ABB RobotStudio station: Estacio120_ROBOTARI_G9.rspag

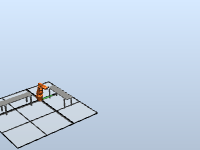
--- station ---
Station Estacio120_ROBOTARI_1415 (saved by RobotStudio format 3)
Controller Sistema120_LEGO_CLOT
  mechanical unit ROB_1: IRB120_3_58__01, 6 joints, base frame (0, 0, 0) mm
Layout (positions relative to the parent item):
  - IRB120_3_58__01 [mechanism, from Robots\IRB120_3_58__01.rslib] at (0, 0, 0) mm; joint values [0.119, 0.2462, -0.2116, 0.435, 0.1998, -0.6575] (rad or m)
  - VENTOSA [mechanism] at (436.31, 58.24, 595.96) mm, rotated rx -12.13 ry 12.35 rz 11.73 deg
      TCP VENTOSA at (0, 0, 0) mm
      links: Conjunto ventosa-muñon
  - Cinta_1 [part] at (0, -1110, 367) mm, rotated rx 0 ry 0 rz 90 deg
  - CINTA2 [part] at (575, 475, 400) mm
Attachment: VENTOSA is attached to IRB120_3_58__01 / Link6
Collision set Conjunto de colisión_1: IRB120_3_58__01, VENTOSA against CINTA2, Cinta_1, near miss 0 m

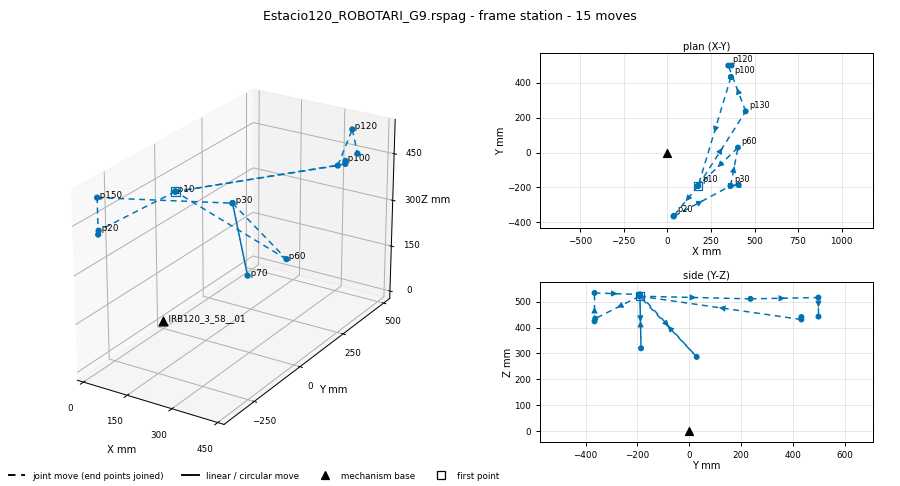
[picture p0: tool path of Estacio120_ROBOTARI_G9.rspag in frame station, 15 of 19 moves have a stored position in this frame; points joined in program order, loops and branches not executed]
--- Backups/Sistema120_LEGO_CLOT/RAPID/TASK1/PROGMOD/CalibData.mod ---
MODULE CalibData
	PERS tooldata VENTOSA:=[TRUE,[[0,0,0],[0.707106781,0,-0.707106781,0]],[0.2,[-60,47,25],[1,0,0,0],0,0,0]];
	TASK PERS tooldata Toolventosa_1:=[TRUE,[[70,0,40],[0.707106781,0,-0.707106781,0]],[0.2,[10,20,10],[1,0,0,0],0,0,0]];
ENDMODULE

--- Backups/Sistema120_LEGO_CLOT/RAPID/TASK1/PROGMOD/MainModule.mod ---
MODULE MainModule

    CONST jointtarget jpos10:=[[6.81954,14.1088,-12.1243,24.9211,11.4493,-37.6717],[9E+09,9E+09,9E+09,9E+09,9E+09,9E+09]];
	CONST robtarget p10:=[[176.81,-191.57,521.21],[0.278921,-0.372832,-0.862871,-0.196606],[-1,0,-1,0],[9E+09,9E+09,9E+09,9E+09,9E+09,9E+09]];
	CONST robtarget p20:=[[36.45,-363.29,434.61],[0.151188,-0.68875,-0.66446,-0.247506],[-1,0,-1,1],[9E+09,9E+09,9E+09,9E+09,9E+09,9E+09]];
	CONST robtarget p30:=[[362.93,-190.78,527.78],[0.208623,-0.296741,-0.924245,-0.119128],[-1,0,-1,1],[9E+09,9E+09,9E+09,9E+09,9E+09,9E+09]];
	CONST robtarget p40:=[[403.50,-186.18,39.16],[0.220229,-0.193089,-0.950068,-0.107642],[-1,-1,0,1],[9E+09,9E+09,9E+09,9E+09,9E+09,9E+09]];
	CONST robtarget p50:=[[405.19,32.89,41.83],[0.208965,-0.192578,-0.952954,-0.105477],[0,0,0,1],[9E+09,9E+09,9E+09,9E+09,9E+09,9E+09]];
	CONST robtarget p60:=[[405.02,28.65,286.65],[0.210569,-0.192705,-0.952533,-0.105863],[0,0,-1,1],[9E+09,9E+09,9E+09,9E+09,9E+09,9E+09]];
	CONST robtarget p70:=[[408.73,-186.25,320.05],[0.21057,-0.192707,-0.952533,-0.105858],[-1,-1,0,1],[9E+09,9E+09,9E+09,9E+09,9E+09,9E+09]];
	CONST robtarget p80:=[[182.80,243.44,681.59],[0.239987,0.420452,-0.872058,0.0716986],[0,0,-1,0],[9E+09,9E+09,9E+09,9E+09,9E+09,9E+09]];
	CONST robtarget p90:=[[364.78,432.80,431.28],[0.29221,0.277543,-0.915161,-0.00793556],[0,-2,1,0],[9E+09,9E+09,9E+09,9E+09,9E+09,9E+09]];
	CONST robtarget p100:=[[364.79,432.79,440.77],[0.292242,0.277494,-0.915166,-0.00792924],[0,-2,1,0],[9E+09,9E+09,9E+09,9E+09,9E+09,9E+09]];
	CONST robtarget p110:=[[368.76,498.78,442.48],[0.292218,0.277507,-0.91517,-0.00789908],[0,-2,1,0],[9E+09,9E+09,9E+09,9E+09,9E+09,9E+09]];
	CONST robtarget p120:=[[349.63,498.54,515.95],[0.262768,0.480674,-0.835673,0.0394526],[0,0,-1,0],[9E+09,9E+09,9E+09,9E+09,9E+09,9E+09]];
	CONST robtarget p130:=[[449.31,236.18,510.99],[0.369937,0.152754,-0.914397,0.0607572],[0,-1,0,0],[9E+09,9E+09,9E+09,9E+09,9E+09,9E+09]];
    CONST robtarget p140:=[[36.47,-365.92,423.85],[0.138204,-0.694353,-0.66549,-0.236425],[-1,0,-1,1],[9E+09,9E+09,9E+09,9E+09,9E+09,9E+09]];
   	CONST robtarget p150:=[[36.44,-365.93,533.78],[0.138198,-0.694384,-0.665464,-0.236409],[-1,0,-1,1],[9E+09,9E+09,9E+09,9E+09,9E+09,9E+09]];
   	LOCAL VAR num Fila_COM1:=0;
   	LOCAL VAR num Columna_COM1:=0;
   	LOCAL VAR num Fila_COM2:=0;
    LOCAL VAR num Columna_COM2:=0;
   	LOCAL VAR bool COM:=False;
    LOCAL VAR bool Peça:=False;
    LOCAL VAR bool Primera_peça:=False;



 PROC  COMANDA(num Columna,num Fila,bool COM)

     FOR Files FROM 0 TO Fila DO

         FOR Columnes FROM 0 TO Columna DO

             IF COM=TRUE THEN

                    MoveJ Offs (p50,(Fila*37.5),(Columna*37.5),0), v1000, fine, tool_ventosa;

             ELSEIF  COM=FALSE THEN

                    MoveJ Offs (p40,(Fila*37.5),(Columna*37.5),0), v1000, fine, tool_ventosa;
             ENDIF
     ENDFOR
        ENDFOR
 ENDPROC



	PROC main()

   !Reset DO10_3;
   SetDO DO10_1,1;  !Activar el compressor
   !POSICIO DE INICI
     MoveAbsJ jpos10\NoEOffs, v1000, z50, tool_ventosa;



 !Espera ordre de final de cicle------------------------------------------------------------------------------------
    IF DI10_4=1 OR Primera_peça=False THEN

     WaitDI DI10_1,1;
     !POSICIO DE LA CINTA 1 ON ESTA LA PEÇA
     MoveJ p10, v1000, z0, tool_ventosa;
     MoveJ p20, v1000, z0, tool_ventosa;
     SetDO DO10_2,1;
     Reset DO10_3;
     MoveJ p140, v1000, z0, tool_ventosa;
     MoveJ p150, v1000, fine, tool_ventosa;
     Peça:=True;
     Primera_peça:=FALSE;

    ENDIF
!Ordre al robot enviar peça a la Comanda 1------------------------------------------------------------------------------------

   IF DI10_2=0 AND  DI10_3=0 AND Peça  THEN      !00

    COM:=False;

   IF Columna_COM1>4 THEN
    Add Fila_COM1,1;
    Columna_COM1:=0;
    ENDIF

    IF Fila_COM1>4 THEN
       Fila_COM1:=0;
    ENDIF

   MoveJ p30, v1000, z0, tool_ventosa;
   MoveJ p70, v1000, z0, tool_ventosa;
   !POSICIO DE LA COMANDA 1
   COMANDA Columna_COM1,Fila_COM1,COM;
   Add Columna_COM1,1;
   Reset DO10_2;
   SetDO DO10_3,1;
   Peça:=False;

   ENDIF

!Ordre al robot enviar peça a la Comanda 2------------------------------------------------------------------------------------

    IF  DI10_2=0 AND  DI10_3=1 AND Peça THEN         !01

    COM:=True;
    IF Columna_COM2>4 THEN
       Add Fila_COM2,1;
       Columna_COM2:=0;
    ENDIF

     IF Fila_COM2>4 THEN
       Fila_COM2:=0;
    ENDIF

    MoveJ p30, v1000, z0, tool_ventosa;
    MoveJ p60, v1000, z0, tool_ventosa;
    !POSICIO DE LA COMANDA 2
    COMANDA Columna_COM2,Fila_COM2,COM;
    Add Columna_COM2,1;
    Reset DO10_2;
    SetDO DO10_3,1;
    Peça:=False;

    ENDIF

!Ordre al robot enviar peça a la cinta 2 a la primera posició------------------------------------------------------------------------------------

    IF  DI10_2=1 AND DI10_3=0 AND Peça THEN        !10
        !POSICIO DEL MAGATZEM 1-2
        MoveJ p10, v1000, z0, tool_ventosa;
        MoveAbsJ jpos10\NoEOffs, v1000, z50, tool_ventosa;
        MoveJ p100, v1000, z0, tool_ventosa;
        MoveL p90, v1000, z0, tool_ventosa;
        Reset DO10_2;
        SetDO DO10_3,1;
        Peça:=False;
        Primera_peça:=True;

    ENDIF

!Ordre al robot enviar peça a la cinta 2 a la segona posició------------------------------------------------------------------------------------

    IF  DI10_2=1 AND  DI10_3=1 AND Peça THEN            !11
        !POSICIO DEL MAGATZEM 3-4
         MoveJ p10, v1000, z0, tool_ventosa;
         MoveJ p130, v1000, z0, tool_ventosa;
         MoveJ p120, v1000, z0, tool_ventosa;
         MoveJ p110, v1000, z0, tool_ventosa;
        Reset DO10_2;
        SetDO DO10_3,1;
        Peça:=False;
        Primera_peça:=True;

    ENDIF



	ENDPROC
ENDMODULE

--- Backups/Sistema120_LEGO_CLOT/HOME/NewProgramName/MainModule.mod ---
MODULE MainModule
	PROC main()

	ENDPROC
ENDMODULE

--- Backups/Sistema120_LEGO_CLOT/SYSPAR/EIO.cfg ---
EIO:CFG_1.0:5:0::
#
EIO_BUS:

      -Name "Virtual1" -ConnectorID "SIM1"

      -Name "DeviceNet1" -BusType "DNET" -ConnectorID "PCI1"\
      -ConnectorLabel "First DeviceNet"

      -Name "DeviceNet_Lean" -BusType "DNLE" -ConnectorID "PCI1"\
      -ConnectorLabel "DeviceNet Lean"

      -Name "Profinet1" -BusType "PNET" -ConnectorID "PCI1"
#
EIO_UNIT_TYPE:

      -Name "Virtual" -VendorName "ABB" -ProductName "Virtual unit"

      -Name "DN_GENERIC" -BusType "DNET" -DN_ExplicitMsgEnabled \
      -DN_C1OutputSize -1 -DN_C1InputSize -1

      -Name "d320" -BusType "DNET" -VendorName "ABB Robotics"\
      -ProductName "120 Vac Unit" -DN_VendorId 75 -DN_ProductCode 1\
      -DN_DeviceType 7 -DN_MajorRev 1 -DN_ExplicitMsgEnabled  -DN_C1Interval 50\
      -DN_C1OutputSize 2 -DN_C1InputSize 2

      -Name "d327A" -BusType "DNET" -VendorName "ABB Robotics"\
      -ProductName "Combi Unit" -DN_VendorId 75 -DN_ProductCode 2\
      -DN_DeviceType 100 -DN_MajorRev 5 -DN_ExplicitMsgEnabled  -DN_C1Type "COS"\
      -DN_C1OutputSize 6 -DN_C1InputSize 2

      -Name "d328A" -BusType "DNET" -VendorName "ABB Robotics"\
      -ProductName "24 VDC Unit" -DN_VendorId 75 -DN_ProductCode 3\
      -DN_DeviceType 7 -DN_ExplicitMsgEnabled  -DN_C1Type "COS"\
      -DN_C1OutputSize 2 -DN_C1InputSize 2

      -Name "d332A" -BusType "DNET" -VendorName "ABB Robotics"\
      -ProductName "Relay Unit" -DN_VendorId 75 -DN_ProductCode 5\
      -DN_DeviceType 7 -DN_MajorRev 2 -DN_ExplicitMsgEnabled  -DN_C1Type "COS"\
      -DN_C1OutputSize 2 -DN_C1InputSize 2

      -Name "d355A" -BusType "DNET" -VendorName "ABB Robotics"\
      -ProductName "Analog Unit" -DN_VendorId 75 -DN_ProductCode 10\
      -DN_DeviceType 100 -DN_MajorRev 1 -DN_ExplicitMsgEnabled \
      -DN_C1Interval 50 -DN_C1OutputSize 8 -DN_C1InputSize 8

      -Name "d651" -BusType "DNET" -VendorName "ABB Robotics"\
      -ProductName "Combi Unit" -DN_VendorId 75 -DN_ProductCode 25\
      -DN_DeviceType 100 -DN_ExplicitMsgEnabled  -DN_C1Type "COS"\
      -DN_C1OutputSize 5 -DN_C1InputSize 1

      -Name "d652" -BusType "DNET" -VendorName "ABB Robotics"\
      -ProductName "24 VDC Unit" -DN_VendorId 75 -DN_ProductCode 26\
      -DN_DeviceType 7 -DN_ExplicitMsgEnabled  -DN_C1Type "COS"\
      -DN_C1OutputSize 2 -DN_C1InputSize 2

      -Name "d653" -BusType "DNET" -VendorName "ABB Robotics"\
      -ProductName "Relay Unit" -DN_VendorId 75 -DN_ProductCode 27\
      -DN_DeviceType 7 -DN_ExplicitMsgEnabled  -DN_C1Type "COS"\
      -DN_C1OutputSize 1 -DN_C1InputSize 1

      -Name "DN_SLAVE" -BusType "DNET" -VendorName "ABB Robotics" -DN_VendorId 8\
      -DN_ProductCode 12 -DN_DeviceType 12 -DN_ExplicitMsgEnabled \
      -DN_C1Interval 50 -DN_C1OutputSize 8 -DN_C1InputSize 8

      -Name "DN_INTERNAL_SLAVE" -BusType "DNET" -VendorName "ABB Robotics"\
      -ProductName "Internal DeviceNet Slave" -InternalSlave  -DN_C1OutputSize 8\
      -DN_C1InputSize 8

      -Name "d350B" -BusType "DNET" -VendorName "ABB Robotics"\
      -ProductName "RIO Adapter" -DN_VendorId 75 -DN_ProductCode 6\
      -DN_DeviceType 7 -DN_MajorRev 2 -DN_ExplicitMsgEnabled  -DN_C1Type "COS"\
      -DN_C1OutputSize -1 -DN_C1InputSize -1

      -Name "d351A" -BusType "DNET" -VendorName "ABB Robotics"\
      -ProductName "IBS Adapter" -DN_VendorId 75 -DN_ProductCode 7\
      -DN_DeviceType 7 -DN_MajorRev 1 -DN_ExplicitMsgEnabled  -DN_C1Type "COS"\
      -DN_C1OutputSize -1 -DN_C1InputSize -1

      -Name "d352A" -BusType "DNET" -VendorName "ABB Robotics"\
      -ProductName "PBUS Adapter" -DN_VendorId 75 -DN_ProductCode 8\
      -DN_DeviceType 7 -DN_MajorRev 1 -DN_ExplicitMsgEnabled  -DN_C1Type "COS"\
      -DN_C1OutputSize -1 -DN_C1InputSize -1

      -Name "d352B" -BusType "DNET" -VendorName "ABB Robotics"\
      -ProductName "PBUS Adapter" -DN_VendorId 75 -DN_ProductCode 8\
      -DN_DeviceType 7 -DN_MajorRev 1 -DN_ExplicitMsgEnabled  -DN_C1Type "COS"\
      -DN_C1OutputSize -1 -DN_C1InputSize -1

      -Name "d378A" -BusType "DNET" -VendorName "ABB Robotics"\
      -ProductName "CCLink Adapter" -DN_VendorId 75 -DN_ProductCode 17\
      -DN_DeviceType 7 -DN_MajorRev 1 -DN_ExplicitMsgEnabled  -DN_C1Interval 50\
      -DN_C1OutputSize -1 -DN_C1InputSize -1

      -Name "d651_Lean" -BusType "DNLE" -VendorName "ABB Robotics"\
      -ProductName "Combi Unit" -DL_ProductCode 25

      -Name "d652_Lean" -BusType "DNLE" -VendorName "ABB Robotics"\
      -ProductName "24 VDC Unit" -DL_ProductCode 26

      -Name "d653_Lean" -BusType "DNLE" -VendorName "ABB Robotics"\
      -ProductName "Relay Unit" -DL_ProductCode 27

      -Name "AC500_PLC_Lean" -BusType "DNLE" -VendorName "ABB Stotz"\
      -ProductName "AC500 PLC - FPB" -DL_ProductCode 1 -DL_VendorID 760

      -Name "DL_GENERIC" -BusType "DNLE" -DL_ProductCode 3535

      -Name "DL_GENERIC_POLL" -BusType "DNLE" -DL_ProductCode 3535\
      -DL_Pollrate 30

      -Name "d351_Lean" -BusType "DNLE" -VendorName "ABB Robotics"\
      -ProductName "IBS Adapter" -DL_ProductCode 7

      -Name "d352_Lean" -BusType "DNLE" -VendorName "ABB Robotics"\
      -ProductName "PBUS Adapter" -DL_ProductCode 8

      -Name "d378_Lean" -BusType "DNLE" -VendorName "ABB Robotics"\
      -ProductName "CCLink Adapter" -DL_ProductCode 17

      -Name "PN_GENERIC" -BusType "PNET" -ProductName "Profinet Device"

      -Name "PN_INTERNAL_SLAVE" -BusType "PNET" -VendorName "ABB Robotics"\
      -ProductName "Internal Profinet Slave" -InternalSlave
#
EIO_UNIT:

      -Name "D652_10" -UnitType "d652" -Bus "DeviceNet1" -DN_Address 10
#
EIO_SIGNAL:

      -Name "DI10_1" -SignalType "DI" -Unit "D652_10" -UnitMap "0"

      -Name "DI10_2" -SignalType "DI" -Unit "D652_10" -UnitMap "1"

      -Name "DI10_3" -SignalType "DI" -Unit "D652_10" -UnitMap "2"

      -Name "DI10_4" -SignalType "DI" -Unit "D652_10" -UnitMap "3"

      -Name "DI10_5" -SignalType "DI" -Unit "D652_10" -UnitMap "4"

      -Name "DI10_6" -SignalType "DI" -Unit "D652_10" -UnitMap "5"

      -Name "DI10_7" -SignalType "DI" -Unit "D652_10" -UnitMap "6"

      -Name "DI10_8" -SignalType "DI" -Unit "D652_10" -UnitMap "7"

      -Name "DI10_9" -SignalType "DI" -Unit "D652_10" -UnitMap "8"

      -Name "DI10_10" -SignalType "DI" -Unit "D652_10" -UnitMap "9"

      -Name "DI10_11" -SignalType "DI" -Unit "D652_10" -UnitMap "10"

      -Name "DI10_12" -SignalType "DI" -Unit "D652_10" -UnitMap "11"

      -Name "DI10_13" -SignalType "DI" -Unit "D652_10" -UnitMap "12"

      -Name "DI10_14" -SignalType "DI" -Unit "D652_10" -UnitMap "13"

      -Name "DI10_15" -SignalType "DI" -Unit "D652_10" -UnitMap "14"

      -Name "DI10_16" -SignalType "DI" -Unit "D652_10" -UnitMap "15"

      -Name "DO10_1" -SignalType "DO" -Unit "D652_10" -UnitMap "0"

      -Name "DO10_2" -SignalType "DO" -Unit "D652_10" -UnitMap "1"

      -Name "DO10_3" -SignalType "DO" -Unit "D652_10" -UnitMap "2"

      -Name "DO10_4" -SignalType "DO" -Unit "D652_10" -UnitMap "3"

      -Name "DO10_5" -SignalType "DO" -Unit "D652_10" -UnitMap "4"

      -Name "DO10_6" -SignalType "DO" -Unit "D652_10" -UnitMap "5"

      -Name "DO10_7" -SignalType "DO" -Unit "D652_10" -UnitMap "6"

      -Name "DO10_8" -SignalType "DO" -Unit "D652_10" -UnitMap "7"

      -Name "DO10_9" -SignalType "DO" -Unit "D652_10" -UnitMap "8"

      -Name "DO10_10" -SignalType "DO" -Unit "D652_10" -UnitMap "9"

      -Name "DO10_11" -SignalType "DO" -Unit "D652_10" -UnitMap "10"

      -Name "DO10_12" -SignalType "DO" -Unit "D652_10" -UnitMap "11"

      -Name "DO10_13" -SignalType "DO" -Unit "D652_10" -UnitMap "12"

      -Name "DO10_14" -SignalType "DO" -Unit "D652_10" -UnitMap "13"

      -Name "DO10_15" -SignalType "DO" -Unit "D652_10" -UnitMap "14"

      -Name "DO10_16" -SignalType "DO" -Unit "D652_10" -UnitMap "15"
#
EIO_COMMAND_TYPE:

      -Name "LinkAddr" -UnitType "d350B" -DefValue "1" -OrderNr 1\
      -DN_Path "6,20 64 24 01 30 01,C6,1" -DN_Service 16

      -Name "DataRate" -UnitType "d350B" -DefValue "0" -OrderNr 2\
      -DN_Path "6,20 64 24 01 30 02,C6,1" -DN_Service 16

      -Name "StartQ" -UnitType "d350B" -DefValue "0" -OrderNr 3\
      -DN_Path "6,20 64 24 01 30 03,C6,1" -DN_Service 16

      -Name "RackSize" -UnitType "d350B" -DefValue "0" -OrderNr 4\
      -DN_Path "6,20 64 24 01 30 04,C6,1" -DN_Service 16

      -Name "LastRack" -UnitType "d350B" -DefValue "0" -OrderNr 5\
      -DN_Path "6,20 64 24 01 30 05,C1,1" -DN_Service 16

      -Name "D350Breset" -UnitType "d350B" -DefValue "0" -OrderNr 6\
      -DN_Path "4,20 01 24 01,C1,1" -DN_Service 5

      -Name "DataWidth" -UnitType "d351A" -DefValue "3" -OrderNr 1\
      -DN_Path "6,20 65 24 01 30 01,C6,1" -DN_Service 16

      -Name "D351Areset" -UnitType "d351A" -DefValue "0" -OrderNr 2\
      -DN_Path "4,20 01 24 01,C1,1" -DN_Service 5

      -Name "MasterInputSize" -UnitType "d352A" -DefValue "1" -OrderNr 1\
      -DN_Path "6,20 67 24 01 30 02,C6,1" -DN_Service 16

      -Name "MasterOutputSize" -UnitType "d352A" -DefValue "1" -OrderNr 2\
      -DN_Path "6,20 67 24 01 30 03,C6,1" -DN_Service 16

      -Name "StationAddress" -UnitType "d352A" -DefValue "126" -OrderNr 3\
      -DN_Path "6,20 67 24 01 30 04,C6,1" -DN_Service 16

      -Name "D352Areset" -UnitType "d352A" -DefValue "0" -OrderNr 4\
      -DN_Path "4,20 01 24 01,C1,1" -DN_Service 5

      -Name "MasterInputSize_B" -UnitType "d352B" -DefValue "1" -OrderNr 1\
      -DN_Path "6,20 67 24 01 30 02,C6,1" -DN_Service 16

      -Name "MasterOutputSize_B" -UnitType "d352B" -DefValue "1" -OrderNr 2\
      -DN_Path "6,20 67 24 01 30 03,C6,1" -DN_Service 16

      -Name "StationAddress_B" -UnitType "d352B" -DefValue "126" -OrderNr 3\
      -DN_Path "6,20 67 24 01 30 04,C6,1" -DN_Service 16

      -Name "D352Breset" -UnitType "d352B" -DefValue "0" -OrderNr 4\
      -DN_Path "4,20 01 24 01,C1,1" -DN_Service 5

      -Name "StationNo" -UnitType "d378A" -DefValue "1" -OrderNr 1\
      -DN_Path "6,20 68 24 01 30 01,C6,1" -DN_Service 16

      -Name "BaudRate" -UnitType "d378A" -DefValue "0" -OrderNr 2\
      -DN_Path "6,20 68 24 01 30 02,C6,1" -DN_Service 16

      -Name "OccStat" -UnitType "d378A" -DefValue "1" -OrderNr 3\
      -DN_Path "6,20 68 24 01 30 03,C6,1" -DN_Service 16

      -Name "BasicIO" -UnitType "d378A" -DefValue "0" -OrderNr 4\
      -DN_Path "6,20 68 24 01 30 04,C1,1" -DN_Service 16

      -Name "D378Areset" -UnitType "d378A" -DefValue "0" -OrderNr 5\
      -DN_Path "4,20 01 24 01,C1,1" -DN_Service 5

      -Name "DataWidth_L" -UnitType "d351_Lean" -DefValue "3" -OrderNr 1\
      -DL_Path "6,20 65 24 01 30 01,C6,1" -DL_Service 16

      -Name "D351reset_L" -UnitType "d351_Lean" -DefValue "0" -OrderNr 2\
      -DL_Path "4,20 01 24 01,C1,1" -DL_Service 5

      -Name "MasterInputSize_B_L" -UnitType "d352_Lean" -DefValue "1" -OrderNr 1\
      -DL_Path "6,20 67 24 01 30 02,C6,1" -DL_Service 16

      -Name "MasterOutputSize_B_L" -UnitType "d352_Lean" -DefValue "1"\
      -OrderNr 2 -DL_Path "6,20 67 24 01 30 03,C6,1" -DL_Service 16

      -Name "StationAddress_B_L" -UnitType "d352_Lean" -DefValue "126"\
      -OrderNr 3 -DL_Path "6,20 67 24 01 30 04,C6,1" -DL_Service 16

      -Name "D352reset_L" -UnitType "d352_Lean" -DefValue "0" -OrderNr 4\
      -DL_Path "4,20 01 24 01,C1,1" -DL_Service 5

      -Name "StationNo_L" -UnitType "d378_Lean" -DefValue "1" -OrderNr 1\
      -DL_Path "6,20 68 24 01 30 01,C6,1" -DL_Service 16

      -Name "BaudRate_L" -UnitType "d378_Lean" -DefValue "0" -OrderNr 2\
      -DL_Path "6,20 68 24 01 30 02,C6,1" -DL_Service 16

      -Name "OccStat_L" -UnitType "d378_Lean" -DefValue "1" -OrderNr 3\
      -DL_Path "6,20 68 24 01 30 03,C6,1" -DL_Service 16

      -Name "BasicIO_L" -UnitType "d378_Lean" -DefValue "0" -OrderNr 4\
      -DL_Path "6,20 68 24 01 30 04,C1,1" -DL_Service 16

      -Name "D378reset_L" -UnitType "d378_Lean" -DefValue "0" -OrderNr 5\
      -DL_Path "4,20 01 24 01,C1,1" -DL_Service 5
#
EIO_ACCESS:

      -Name "All" -Rapid  -LocalManual  -LocalAuto  -RemoteManual  -RemoteAuto
